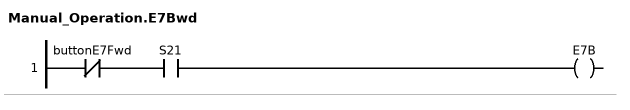
[picture p24: Manual_Operation.E7Bwd (LD)]
_LD_ (* Ladder Diagram *)
NETWORK 1
	[/buttonE7Fwd] - [S21] --- (E7B)
_END_LD_
(* the same logic as Structured Text *)
(* Network 1 *)
E7B := NOT buttonE7Fwd AND S21;
END_ACTION
ACTION E8Bwd:
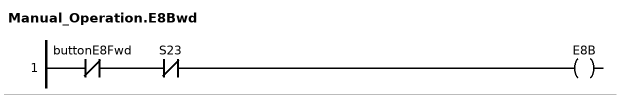
_LD_ (* Ladder Diagram *)
NETWORK 1
	[/buttonE8Fwd] - [/S23] --- (E8B)
_END_LD_
(* the same logic as Structured Text *)
(* Network 1 *)
E8B := NOT buttonE8Fwd AND NOT S23;
END_ACTION
ACTION E8Fwd:
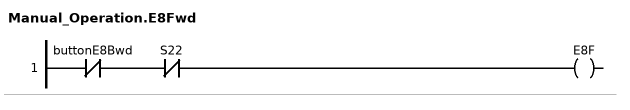
_LD_ (* Ladder Diagram *)
NETWORK 1
	[/buttonE8Bwd] - [/S22] --- (E8F)
_END_LD_
(* the same logic as Structured Text *)
(* Network 1 *)
E8F := NOT buttonE8Bwd AND NOT S22;
END_ACTION
ACTION E9Down:
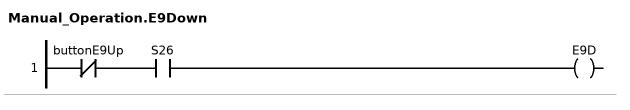
_LD_ (* Ladder Diagram *)
NETWORK 1
	[/buttonE9Up] - [S26] --- (E9D)
_END_LD_
(* the same logic as Structured Text *)
(* Network 1 *)
E9D := NOT buttonE9Up AND S26;
END_ACTION
ACTION E9Up:
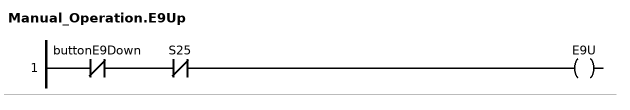
_LD_ (* Ladder Diagram *)
NETWORK 1
	[/buttonE9Down] - [/S25] --- (E9U)
_END_LD_
(* the same logic as Structured Text *)
(* Network 1 *)
E9U := NOT buttonE9Down AND NOT S25;
END_ACTION

(* POU Automatic_Operation, SFC *)
PROGRAM Automatic_Operation
VAR
END_VAR
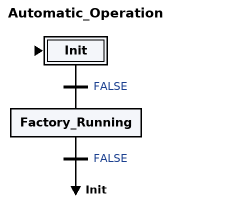
INITIAL_STEP Init:
END_STEP
TRANSITION FROM Init TO Factory_Running := FALSE;
END_TRANSITION
STEP Factory_Running:
END_STEP
TRANSITION FROM Factory_Running TO Init := FALSE;
END_TRANSITION
END_PROGRAM

(* POU Automatic_Conditional, LD *)
PROGRAM Automatic_Conditional
VAR
END_VAR
_LD_ (* Ladder Diagram *)
_END_LD_
END_PROGRAM

(* POU Base_Storage, SFC *)
PROGRAM Base_Storage
VAR
END_VAR
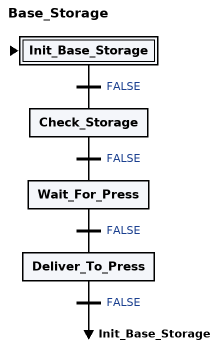
INITIAL_STEP Init_Base_Storage:
END_STEP
TRANSITION FROM Init_Base_Storage TO Check_Storage := FALSE;
END_TRANSITION
STEP Check_Storage:
END_STEP
TRANSITION FROM Check_Storage TO Wait_For_Press := FALSE;
END_TRANSITION
STEP Wait_For_Press:
END_STEP
TRANSITION FROM Wait_For_Press TO Deliver_To_Press := FALSE;
END_TRANSITION
STEP Deliver_To_Press:
END_STEP
TRANSITION FROM Deliver_To_Press TO Init_Base_Storage := FALSE;
END_TRANSITION
END_PROGRAM

(* POU Press, SFC *)
PROGRAM Press
VAR
END_VAR
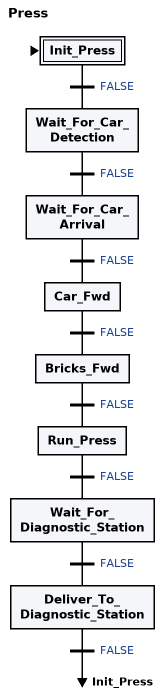
INITIAL_STEP Init_Press:
END_STEP
TRANSITION FROM Init_Press TO Wait_For_Car_Detection := FALSE;
END_TRANSITION
STEP Wait_For_Car_Detection:
END_STEP
TRANSITION FROM Wait_For_Car_Detection TO Wait_For_Car_Arrival := FALSE;
END_TRANSITION
STEP Wait_For_Car_Arrival:
END_STEP
TRANSITION FROM Wait_For_Car_Arrival TO Car_Fwd := FALSE;
END_TRANSITION
STEP Car_Fwd:
END_STEP
TRANSITION FROM Car_Fwd TO Bricks_Fwd := FALSE;
END_TRANSITION
STEP Bricks_Fwd:
END_STEP
TRANSITION FROM Bricks_Fwd TO Run_Press := FALSE;
END_TRANSITION
STEP Run_Press:
END_STEP
TRANSITION FROM Run_Press TO Wait_For_Diagnostic_Station := FALSE;
END_TRANSITION
STEP Wait_For_Diagnostic_Station:
END_STEP
TRANSITION FROM Wait_For_Diagnostic_Station TO Deliver_To_Diagnostic_Station := FALSE;
END_TRANSITION
STEP Deliver_To_Diagnostic_Station:
END_STEP
TRANSITION FROM Deliver_To_Diagnostic_Station TO Init_Press := FALSE;
END_TRANSITION
END_PROGRAM

(* POU Diagnostic_Station, SFC *)
PROGRAM Diagnostic_Station
VAR
END_VAR
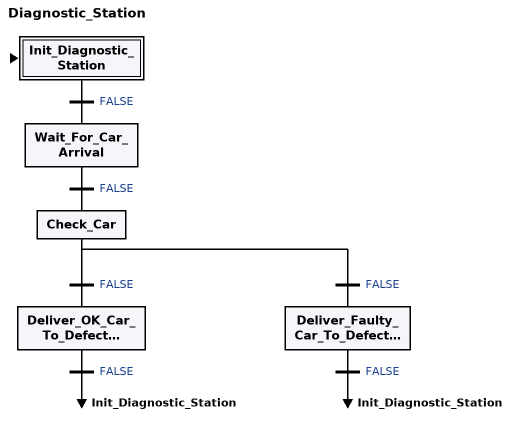
INITIAL_STEP Init_Diagnostic_Station:
END_STEP
TRANSITION FROM Init_Diagnostic_Station TO Wait_For_Car_Arrival := FALSE;
END_TRANSITION
STEP Wait_For_Car_Arrival:
END_STEP
TRANSITION FROM Wait_For_Car_Arrival TO Check_Car := FALSE;
END_TRANSITION
STEP Check_Car:
END_STEP
TRANSITION FROM Check_Car TO Deliver_OK_Car_To_Defect_Separation := FALSE;
END_TRANSITION
TRANSITION FROM Check_Car TO Deliver_Faulty_Car_To_Defect_Separation := FALSE;
END_TRANSITION
STEP Deliver_OK_Car_To_Defect_Separation:
END_STEP
TRANSITION FROM Deliver_OK_Car_To_Defect_Separation TO Init_Diagnostic_Station := FALSE;
END_TRANSITION
STEP Deliver_Faulty_Car_To_Defect_Separation:
END_STEP
TRANSITION FROM Deliver_Faulty_Car_To_Defect_Separation TO Init_Diagnostic_Station := FALSE;
END_TRANSITION
END_PROGRAM

(* POU Defect_Separation, SFC *)
PROGRAM Defect_Separation
VAR
END_VAR
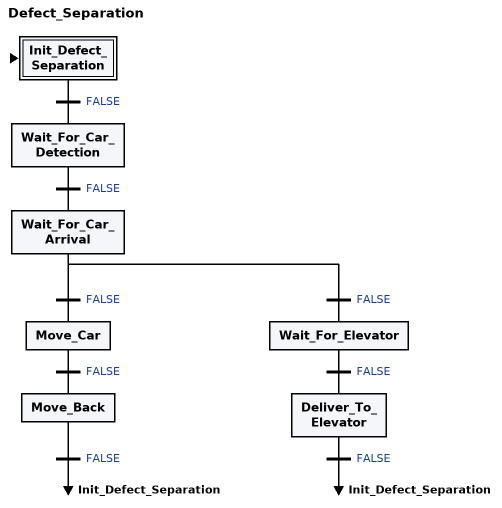
INITIAL_STEP Init_Defect_Separation:
END_STEP
TRANSITION FROM Init_Defect_Separation TO Wait_For_Car_Detection := FALSE;
END_TRANSITION
STEP Wait_For_Car_Detection:
END_STEP
TRANSITION FROM Wait_For_Car_Detection TO Wait_For_Car_Arrival := FALSE;
END_TRANSITION
STEP Wait_For_Car_Arrival:
END_STEP
TRANSITION FROM Wait_For_Car_Arrival TO Move_Car := FALSE;
END_TRANSITION
TRANSITION FROM Wait_For_Car_Arrival TO Wait_For_Elevator := FALSE;
END_TRANSITION
STEP Move_Car:
END_STEP
TRANSITION FROM Move_Car TO Move_Back := FALSE;
END_TRANSITION
STEP Move_Back:
END_STEP
TRANSITION FROM Move_Back TO Init_Defect_Separation := FALSE;
END_TRANSITION
STEP Wait_For_Elevator:
END_STEP
TRANSITION FROM Wait_For_Elevator TO Deliver_To_Elevator := FALSE;
END_TRANSITION
STEP Deliver_To_Elevator:
END_STEP
TRANSITION FROM Deliver_To_Elevator TO Init_Defect_Separation := FALSE;
END_TRANSITION
END_PROGRAM

(* POU Elevator, SFC *)
PROGRAM Elevator
VAR
END_VAR
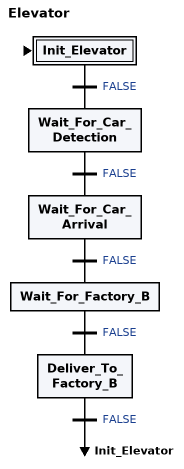
INITIAL_STEP Init_Elevator:
END_STEP
TRANSITION FROM Init_Elevator TO Wait_For_Car_Detection := FALSE;
END_TRANSITION
STEP Wait_For_Car_Detection:
END_STEP
TRANSITION FROM Wait_For_Car_Detection TO Wait_For_Car_Arrival := FALSE;
END_TRANSITION
STEP Wait_For_Car_Arrival:
END_STEP
TRANSITION FROM Wait_For_Car_Arrival TO Wait_For_Factory_B := FALSE;
END_TRANSITION
STEP Wait_For_Factory_B:
END_STEP
TRANSITION FROM Wait_For_Factory_B TO Deliver_To_Factory_B := FALSE;
END_TRANSITION
STEP Deliver_To_Factory_B:
END_STEP
TRANSITION FROM Deliver_To_Factory_B TO Init_Elevator := FALSE;
END_TRANSITION
END_PROGRAM
